(* PLC project Pizzarocessor_28_10_2025.project, CODESYS CODESYS V3.5 SP21 Patch 1 *)
(* stored: creationDateTime 2025-11-03T11:35:46.0292408, modificationDateTime 2025-10-30T21:42:08.8139206 *)

TYPE HopperStatus : STRUCT
  Hopper_Id : INT;  (* id for each Hopper *)
  Fill_Level : REAL;  (* percentage of hooper *)
  Ingredient_ID : STRING(20);  (* Ingredient Name *)
  Alarm_Active : BOOL;  (* Alarm *)
  Is_Dispensing : BOOL;  (* Ingredient is being dispensed *)
END_STRUCT;
END_TYPE

TYPE ConveyorStatus : STRUCT
  Conveyor_ID : INT;  (* Conveyor number/ID *)
  Speed : REAL;  (* Percentage of speed *)
  Jam_Detected : BOOL;  (* Conveyor is Jammed *)
  Running : BOOL;
END_STRUCT;
END_TYPE

PROGRAM Supervisor_PRG
  VAR
    b_Mode : BOOL;  (* True = Auto, False = Manual *)
    b_Hopper_Empty : ARRAY[1..5] OF BOOL;  (* 1=Base, 2=Toppings, 3=Oregano, 4=Chilli, 5=Box (if you treat Box similarly) *)
    b_Conveyor_Jam : ARRAY[1..3] OF BOOL;  (* 3 conveyors Jam Status *)
    b_Interlock_Hopper : ARRAY[1..5] OF BOOL;  (* Matches hopper indices *)
    b_Interlock_Conveyor : ARRAY[1..3] OF BOOL;  (* Interlocks for conveyors *)
    b_Interlock_OtherZones : ARRAY[1..2] OF BOOL;  (* Example: 1=HeatingZone, 2=PackingStation *)
    b_Alarm_HopperEmpty : BOOL;  (* Alarm Flags *)
    b_Alarm_ConveyorJam : BOOL;
    i_Jammed_Conveyor_Index : INT;  (* 0 = none, else 1..n conveyor index *)
    i_Empty_Hopper_Index : INT;
    b_Alarm_Reset_Command : BOOL;  (* Command from HMI to reset alarms *)
  END_VAR

                    
                  
END_PROGRAM

FUNCTION_BLOCK FB_Hopper
  VAR_INPUT
    StartDispense : BOOL;
    StopDispense : BOOL;
  END_VAR
  VAR_OUTPUT
    Status : HopperStatus;
  END_VAR
  VAR
    Internal_State : BOOL;  (* False=Idle True= Dispensing *)
  END_VAR

                    //Hopper Control Logic
IF StartDispense THEN
	Status.Is_Dispensing:= TRUE;
	Internal_State := TRUE;
ELSIF StopDispense THEN
	Status.Is_Dispensing:= FALSE;
	Internal_State := FALSE;
END_IF

//Simulate Ingredient level
IF Internal_State =1 THEN
   Status.Fill_Level := Status.Fill_Level - 0.1; // Decrement per Order
END_IF

//Alarm Logic
status.Alarm_Active := (status.Fill_Level < 5.0);
                  
END_FUNCTION_BLOCK

FUNCTION_BLOCK FB_Conveyor
  VAR_INPUT
    Start : BOOL;
    Speed_Setpoint : REAL;  (* percentage in speed *)
  END_VAR
  VAR_OUTPUT
    Running : BOOL;
    Fault : BOOL;
    Jam_Detected : BOOL;
    Current_Speed : REAL;
  END_VAR
  VAR
    State : INT;  (* 0=Ideal, 1=running, 2=Fault *)
  END_VAR

                    // Logic Framework
IF Fault THEN
	Running := FALSE;
	Current_Speed := 0.0;
	State := 2;
ELSE
	IF NOT Fault AND Start = TRUE THEN
	   Running := TRUE;
	   Current_Speed := Speed_Setpoint;
	   State := 1;
	 ELSIF NOT Start THEN 
     	Running := FALSE;
	    Current_Speed := 0.0;
	    State := 0;	
		 
		
		
	END_IF
	
END_IF


	

                  
END_FUNCTION_BLOCK

CONFIGURATION Device
  RESOURCE Application ON PLC
    TASK MainTask(INTERVAL := T#20ms, PRIORITY := 1);
    PROGRAM Supervisor_PRG WITH MainTask : Supervisor_PRG;
  END_RESOURCE
END_CONFIGURATION
